// SIMATIC S7-200 project (STEP 7-Micro/WIN), CPU 224 UN REL 02.02

SYMBOL_TABLE USER1
Start            I0.4
_Stop            I0.5
D1               I0.3
D2               I0.1
D3               I0.2
Conveyer         Q0.4
Heater           Q0.1
Red              Q0.2
Green            Q0.3
END_SYMBOL_TABLE

ORGANIZATION_BLOCK MAIN:OB1
TITLE=PROGRAM COMMENTS
BEGIN
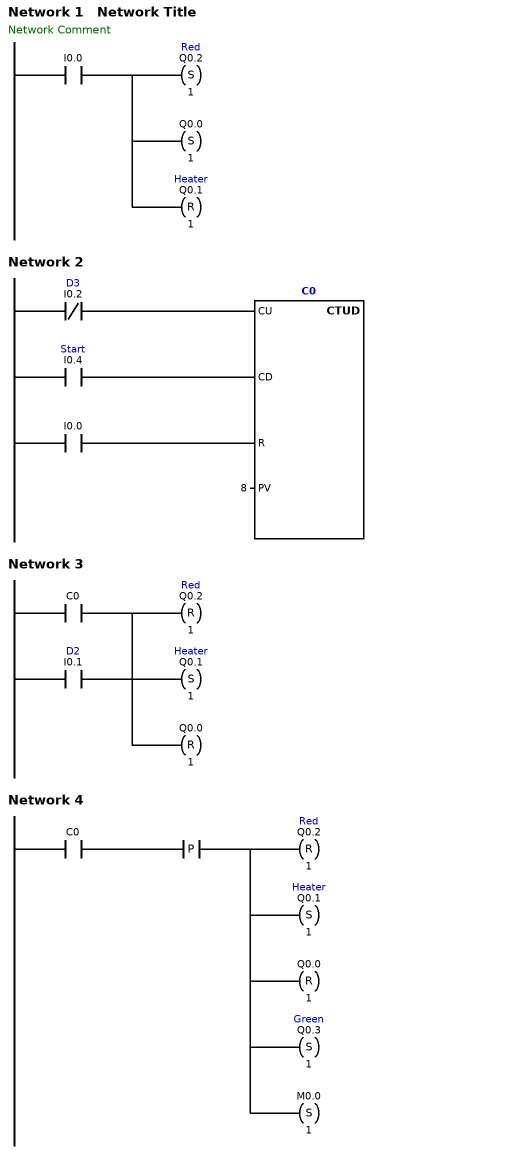
Network 1 //  Network Title
//  Network Comment
LD     I0.0
S      Red:Q0.2, 1
S      Q0.0, 1
R      Heater:Q0.1, 1
Network 2
LDN    D3:I0.2
LD     Start:I0.4
LD     I0.0
CTUD   C0, 8
Network 3
LD     C0
O      D2:I0.1
R      Red:Q0.2, 1
S      Heater:Q0.1, 1
R      Q0.0, 1
Network 4
LD     C0
EU
R      Red:Q0.2, 1
S      Heater:Q0.1, 1
R      Q0.0, 1
S      Green:Q0.3, 1
S      M0.0, 1
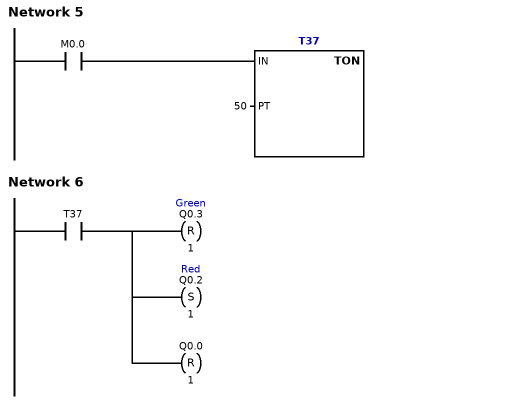
Network 5
LD     M0.0
TON    T37, 50
Network 6
LD     T37
R      Green:Q0.3, 1
S      Red:Q0.2, 1
R      Q0.0, 1
END_ORGANIZATION_BLOCK
